FUNCTION_BLOCK FILLPOLY (* openCV fillPolygon *)
  (* Version 1.0, AN, SWDC RTSoft *)
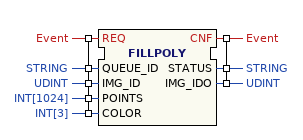
  EVENT_INPUT
    REQ WITH QUEUE_ID, IMG_ID, POINTS, COLOR;
  END_EVENT
  EVENT_OUTPUT
    CNF WITH STATUS, IMG_IDO;
  END_EVENT
  VAR_INPUT
    QUEUE_ID : STRING;
    IMG_ID : UDINT;
    POINTS : ARRAY [0..1023] OF INT;
    COLOR : ARRAY [0..2] OF INT; (* Color of the filled polygon [B, G, R] *)
  END_VAR
  VAR_OUTPUT
    STATUS : STRING;
    IMG_IDO : UDINT;
  END_VAR
  ALGORITHM REQ IN ST:

  END_ALGORITHM
END_FUNCTION_BLOCK
